FUNCTION_BLOCK EM_LiftingTransport EXTENDS EM_Base IMPLEMENTS I_EM_LiftingTransport

VAR_INPUT
//Inputs
	i_ref_stSettings : REFERENCE TO ST_SettingsLiftingTransport;
	
	i_bIlckLiftUp : BOOL := TRUE;
	i_bIlckLiftDown : BOOL := TRUE;
	i_bIlckTransportExtract : BOOL := TRUE;
	i_bIlckTransportRetract : BOOL := TRUE;
	
	i_refTB : REFERENCE TO OBJ_Carrier;	//Mogelijk voor uiteindelijke machine, voor de FUMO's is dit nog niet echt relevant
	
	
	s_arr_bTest : ARRAY[0..15] OF BOOL; 
END_VAR

VAR_OUTPUT
	q_bStaWarning : BOOL;
END_VAR

VAR
	
axisLift : AXIS_REF;
axisTransportUnit : AXIS_REF;

//------------------------------------------//
//Control Modules (Devices)
	s_cmLift : CM_AX5000;
	s_cmTransportUnit : CM_AX5000;
	
//------------------------------------------//

//------------------------------------------//
//Inputs
//------------------------------------------//
	
//------------------------------------------//
//Outputs

//------------------------------------------//

//Requests
{warning '#TODO": Update to Lifting Transport'}
s_bReqTB_ToInfeed : BOOL := FALSE;
s_bReqTB_ToCenter : BOOL := FALSE;
s_bReqTB_ToDocking : BOOL := FALSE;
s_bReqCenteringTB : BOOL := FALSE;

//States
{warning '#TODO": Update to Lifting Transport'}
s_bStaBrakeReleased : BOOL := FALSE;
s_bStaDriveError : BOOL := FALSE;

//Properties
	
//Interlockes	
	s_bIlckLiftUp : BOOL := TRUE;
	s_bIlckLiftDown : BOOL := TRUE;
	s_bIlckTransportExtract : BOOL := TRUE;
	s_bIlckTransportRetract : BOOL := TRUE;
	
	{warning '#TODO: are these variable / properies really nessecary?' }
	s_bStaTB_AtInfeed : BOOL;
	s_bStaTB_AtCentering : BOOL;
	s_bStaTB_AtDocking : BOOL;
	s_bStaTB_CenteringDone : BOOL;
	
	
//Alarms
	s_sReason : STRING;
	{warning '#TODO": Update to Lifting Transport'}
	s_fbAlarmHandlerTravelTimeOut : FB_AlarmHandler;
	s_bErrTravelTimeOut : BOOL;
	
//Warnings
{warning '#TODO": Update to Lifting Transport'}
	s_fbAlarmHandlerOuterDoorNotOpened : FB_AlarmHandler;
	s_bWrnOuterDoorNotOpened : BOOL;
	
	s_bStaWarning : BOOL;
	
//------------------------------------------//
//Params
//--	//Tool settings
//--	s_fbParamToolHardwareNr				: FB_HmiParamHandler;
//--    s_fbParamToolSoftwareVersion		: FB_HmiParamHandler;

//--	s_fbParamName						: FB_HmiParamHandler;
//--	s_fbParamNumber						: FB_HmiParamHandler;
//--	s_fbParamRevision                   : FB_HmiParamHandler;
	
//--	s_fbParamTeslaMeterIp				: FB_HmiParamHandler;
//--	s_fbParamTeslaMeterPort				: FB_HmiParamHandler;
	
//--	//Product settings (Maybe)
//--	s_fbParamTotalStroke				: FB_HmiParamHandler;
//--	s_fbParamStepStroke					: FB_HmiParamHandler;
//--	s_fbParamAveragingNumberTest		: FB_HmiParamHandler;
	
//--	s_fbParamaMaxMagnitudeCriteria		: FB_HmiParamHandler;
	
//--	s_fbParamRefIduBottom				: FB_HmiParamHandler;
//--	s_fbParamRefItm                     : FB_HmiParamHandler;
//--	s_fbParamRefCenterTpmPipe           : FB_HmiParamHandler;
//--	s_fbParamRefCpValve					: FB_HmiParamHandler;
//------------------------------------------//

//------------------------------------------//
//Variables
//--	s_sTestResult 						: STRING;
	
//------------------------------------------//

//------------------------------------------//
//Alarms
	

//------------------------------------------//

//------------------------------------------//

	s_sMessage : STRING;

//Sequencers
	s_eSeqLiftingTransport : E_SeqLiftingTransport;
	s_fbSeqLiftingTransportControl : FB_SeqControl;

	s_eTmpLocation : E_Location;
	s_eTmpCenteringDone : BOOL;
	
	s_tMaxTravelTime : TIME;
	s_tDoorCheckTime : TIME;
	s_bDoorCheckTimeDisabled : BOOL := FALSE;
	

//Hmi
{warning '#TODO": Update to Lifting Transport'}
	s_nToHmiStepNr					: INT;
	s_nToHmiMaxStepNr				: INT;
	s_sToHmiInstructionText			: T_MAXSTRING;
	s_sToHmiProcedure				: T_MAXSTRING;
	
	//Buttons
	s_fbHmiBtnTB_ToInfeed				: FB_HmiBtn;
	s_fbHmiBtnTB_ToCentering			: FB_HmiBtn;
	s_fbHmiBtnTB_ToDocking				: FB_HmiBtn;
	
	s_fbHmiBtnTB_Centering				: FB_HmiBtn;
	
	//Leds
	s_fbHmiLedInfeedRearPosition		: FB_HmiLed;
	s_fbHmiLedInfeedFrontPosition		: FB_HmiLed;
	s_fbHmiLedCenteringPosition			: FB_HmiLed;
	s_fbHmiLedDockingPosition			: FB_HmiLed;
	s_fbHmiLedDoorOpened				: FB_HmiLed;
	
	s_fbHmiLedCenteringIdle				: FB_HmiLed;
	s_fbHmiLedCenteringCenter			: FB_HmiLed;
	
//------------------------------------------//
END_VAR

	
SUPER^();

METHOD PROTECTED _m_Alarms : BOOL

IF NOT SUPER^._m_Alarms() THEN
	RETURN;
END_IF

{warning '#TODO": Update to Lifting Transport'}
// Alarm Handlers
s_fbAlarmHandlerTravelTimeOut(
	i_bStaActive := s_bErrTravelTimeOut, 
	i_eAlarmLevel := E_AlarmLevel.Alarm, 
	i_sAlarmText := CONCAT(i_sEmName, CONCAT( ': Travel error: ', s_sReason)));
	
s_fbAlarmHandlerOuterDoorNotOpened(
	i_bStaActive := s_bWrnOuterDoorNotOpened, 
	i_eAlarmLevel := E_AlarmLevel.Warning, 
	i_sAlarmText := CONCAT(i_sEmName, ': Outer-door open not detected'));

// Reset warnings
IF i_bCmdReset THEN
	s_bErrTravelTimeOut := FALSE;
	s_bWrnOuterDoorNotOpened := FALSE;
END_IF

s_bStaError := 
	s_cmPalletConveyor.p_bStaError
	OR s_cmCenteringUnit.p_bStaError
	OR s_fbAlarmHandlerTravelTimeOut.q_bStaActive;	

s_bStaWarning :=
	s_fbAlarmHandlerOuterDoorNotOpened.q_bStaActive
	OR s_cmPalletConveyor.p_bStaWarning
	OR s_cmCenteringUnit.p_bStaWarning;
	
_m_Alarms := TRUE;
END_METHOD

METHOD PRIVATE _m_AutomaticControl : BOOL

//Lifting Transport
_m_SeqLiftingTransport();
END_METHOD

METHOD PROTECTED _m_Devices : BOOL

IF NOT SUPER^._m_Devices() THEN
	RETURN;
END_IF

s_cmLift(
	i_bReqEnable := i_bReqEnable,
	i_eCtrlMode := i_eCtrlMode,
	i_bCmdReset := i_bCmdReset,
	i_refAxis := axisLift,
	i_bIclkForward := FALSE,
	i_bIclkBackward := FALSE);

s_cmTransportUnit(
	i_bReqEnable := i_bReqEnable,
	i_eCtrlMode := i_eCtrlMode,
	i_bCmdReset := i_bCmdReset,
	i_refAxis := axisTransportUnit,
	i_bIclkForward := FALSE, 
	i_bIclkBackward := FALSE);

_m_Devices := TRUE;
END_METHOD

METHOD PROTECTED _m_Hmi : BOOL

IF NOT SUPER^._m_Hmi() THEN
	RETURN;
END_IF

//Buttons
s_fbHmiBtnTB_ToInfeed.p_bStaEnabled := s_bIlckConveyorBackward;
s_fbHmiBtnTB_ToCentering.p_bStaEnabled := s_bIlckConveyorForward;
s_fbHmiBtnTB_ToDocking.p_bStaEnabled := s_bIlckConveyorForward;
s_fbHmiBtnTB_Centering.p_bStaEnabled := s_bIlckCenteringToCenter;

s_fbHmiBtnTB_ToInfeed();
s_fbHmiBtnTB_ToCentering();
s_fbHmiBtnTB_ToDocking();
s_fbHmiBtnTB_Centering();

//Leds
s_fbHmiLedInfeedRearPosition(i_bStaLed := s_bStaAtInfeedRearPosition);
s_fbHmiLedInfeedFrontPosition(i_bStaLed := s_bStaAtInfeedFrontPosition);
s_fbHmiLedCenteringPosition(i_bStaLed := s_bStaAtCenteringPosition);
s_fbHmiLedDockingPosition(i_bStaLed := s_bStaAtDockingPosition);
s_fbHmiLedDoorOpened(i_bStaLed := s_bStaDoorOpened);

s_fbHmiLedCenteringCenter(i_bStaLed := s_bStaCenteringCenter);
s_fbHmiLedCenteringIdle(i_bStaLed := s_bStaCenteringIdle);

_m_Hmi := TRUE;
END_METHOD

METHOD PROTECTED _m_Init : BOOL

IF NOT SUPER^._m_Init() THEN
	RETURN;
END_IF

//Control Modules
s_cmLift.i_bReqEnable := FALSE;
s_cmLift.i_eCtrlMode := E_CtrlMode.IDLE;
s_cmLift.i_sCmName := 'CM Lift';
s_cmLift.i_refAxis REF= axisLift;

s_cmTransportUnit.i_bReqEnable := FALSE;
s_cmTransportUnit.i_eCtrlMode := E_CtrlMode.IDLE;
s_cmTransportUnit.i_sCmName := 'CM Transport Unit';
s_cmTransportUnit.i_refAxis REF= axisTransportUnit;
{warning '#TODO: Dot we need to added configuration parameters? Seperate struct or via settings or dedicateed variables'}

//---------------------------------//	
	
//----------------------------------//	
//Hmi
{warning '#TODO: Update to Lifing Transport'} 
	s_fbHmiBtnTB_ToInfeed.p_eButtontype := E_HmiButtonType.PUSHBUTTON;
	s_fbHmiBtnTB_ToInfeed.p_bStaVisible := FALSE;
	s_fbHmiBtnTB_ToInfeed.p_bStaEnabled := FALSE;		
	s_fbHmiBtnTB_ToInfeed.p_sBtnText := 'TB To Infeed Position';
	
	s_fbHmiBtnTB_ToCentering.p_eButtontype := E_HmiButtonType.PUSHBUTTON;
	s_fbHmiBtnTB_ToCentering.p_bStaVisible := FALSE;
	s_fbHmiBtnTB_ToCentering.p_bStaEnabled := FALSE;		
	s_fbHmiBtnTB_ToCentering.p_sBtnText := 'TB To Centering Position';
	
	s_fbHmiBtnTB_ToDocking.p_eButtontype := E_HmiButtonType.PUSHBUTTON;
	s_fbHmiBtnTB_ToDocking.p_bStaVisible := FALSE;
	s_fbHmiBtnTB_ToDocking.p_bStaEnabled := FALSE;		
	s_fbHmiBtnTB_ToDocking.p_sBtnText := 'TB To Docking Position';
	
	s_fbHmiBtnTB_Centering.p_eButtontype := E_HmiButtonType.PUSHBUTTON;
	s_fbHmiBtnTB_Centering.p_bStaVisible := FALSE;
	s_fbHmiBtnTB_Centering.p_bStaEnabled := FALSE;		
	s_fbHmiBtnTB_Centering.p_sBtnText := 'Centering TB';

	s_fbHmiLedInfeedRearPosition.p_bStaVisible := FALSE;
	s_fbHmiLedInfeedRearPosition.p_sToHmiDescriptionLed := 'Infeed Rear Position';
	
	s_fbHmiLedInfeedFrontPosition.p_bStaVisible := FALSE;
	s_fbHmiLedInfeedFrontPosition.p_sToHmiDescriptionLed := 'Infeed Front Position';
	
	s_fbHmiLedCenteringPosition.p_bStaVisible := FALSE;
	s_fbHmiLedCenteringPosition.p_sToHmiDescriptionLed := 'Center Position';
	
	s_fbHmiLedDockingPosition.p_bStaVisible := FALSE;
	s_fbHmiLedDockingPosition.p_sToHmiDescriptionLed := 'Docking Position';
	
	s_fbHmiLedDoorOpened.p_bStaVisible := FALSE;
	s_fbHmiLedDoorOpened.p_sToHmiDescriptionLed := 'Door Opened';
	
	s_fbHmiLedCenteringIdle.p_bStaVisible := FALSE;
	s_fbHmiLedCenteringIdle.p_sToHmiDescriptionLed := 'Centering Idle';
	
	s_fbHmiLedCenteringCenter.p_bStaVisible := FALSE;
	s_fbHmiLedCenteringCenter.p_sToHmiDescriptionLed := 'Centering Center';
	
//----------------------------------//	
//Initialize all moving averages

//----------------------------------//	

//----------------------------------//	

//Inputs
//----------------------------------//	

//----------------------------------//	
//Outputs
//--s_doRelayTableDown.i_stSettings.bCfgDelay		:= FALSE;	
//--s_doRelayTableDown.i_stSettings.tmOutputDelay	:= T#0S;	
//----------------------------------//	

_m_Init := TRUE;
END_METHOD

METHOD PROTECTED _m_Inputs : BOOL
IF NOT SUPER^._m_Inputs() THEN
	RETURN;
END_IF

//Interlocks
s_bIlckConveyorForward := i_bIlckConveyorForward OR NOT(s_bStaCenteringIdle); 
s_bIlckConveyorBackward := i_bIlckConveyorBackward OR NOT(s_bStaCenteringIdle);
s_bIlckConveyorBackward := NOT(s_bStaCenteringIdle);
s_bIlckCenteringToCenter := NOT(s_cmPalletConveyor.p_bStaMotorStopped);
s_bIlckCenteringToIdle := FALSE;

//Reasons
IF i_bIlckConveyorForward OR i_bIlckConveyorBackward THEN
	s_cmPalletConveyor.p_sInterlockedReason := 'External interlocked';
ELSIF s_bIlckConveyorForward OR s_bIlckConveyorBackward THEN
	s_cmPalletConveyor.p_sInterlockedReason := 'Centering not in idle-position'; 
END_IF

IF s_bIlckCenteringToCenter THEN
	s_cmCenteringUnit.p_sInterlockedReason := 'Conveyor not stopped';
END_IF

_m_Inputs := TRUE;
END_METHOD

METHOD PRIVATE _m_ManualControl : BOOL

// Manual control has been implemented into lower layer control modules
END_METHOD

METHOD _m_MoveAbsolute : BOOL
VAR_INPUT
	i_ref_axis : REFERENCE TO TC2_MC2.AXIS_REF;
	i_ref_stProfile : ST_PositioningProfile;
END_VAR

VAR_INST
	s_MC_MoveAbsolute : TC2_MC2.MC_MoveAbsolute;
END_VAR

IF NOT(__ISVALIDREF(i_ref_axis)) THEN
	// Message invalid reference
	RETURN;
END_IF

s_MC_MoveAbsolute(
	Axis := i_ref_axis,
	Execute := TRUE AND NOT(s_MC_MoveAbsolute.Busy OR s_MC_MoveAbsolute.Done OR s_MC_MoveAbsolute.Error),
	Position := i_ref_stProfile.fPosition,
	Velocity := i_ref_stProfile.fVelocity,
	Acceleration := i_ref_stProfile.fAcceleration,
	Deceleration := i_ref_stProfile.fDeceleration,
	Jerk := i_ref_stProfile.fJerk,
	BufferMode := TC2_MC2.MC_BufferMode.MC_Aborting,
	Options := ,
	Done => ,
	Busy => ,
	Active => ,
	CommandAborted => ,
	Error => ,
	ErrorID => );
	
_m_MoveAbsolute := s_MC_MoveAbsolute.Done;
END_METHOD

METHOD PROTECTED _m_Outputs : BOOL

IF NOT SUPER^._m_Outputs() THEN
	RETURN;
END_IF

q_bStaWarning := s_bStaWarning;

_m_Outputs := TRUE;
END_METHOD

METHOD PROTECTED _m_Params : BOOL
VAR_INST
	s_fToHmiXAxisMin	: LREAL;
	s_fToHmiXAxisMax	: LREAL;
	s_fToHmiYAxisMin	: LREAL;
	s_fToHmiYAxisMax	: LREAL;
END_VAR

IF NOT SUPER^._m_Params() THEN
	RETURN;
END_IF

s_fbParamToolHardwareNr(i_fDefaultValue				:= 0,
						i_nArrayFolderIndex			:= 1,
						i_sName						:= 'Harware ID',
						i_bIsNumber					:= FALSE);

s_fbParamToolSoftwareVersion(i_fDefaultValue		:= 0,
							i_nArrayFolderIndex		:= 1,
							i_sName					:= 'Software Version',
							i_bIsNumber				:= FALSE);

s_fbParamName(i_fDefaultValue						:= 0,
				i_nArrayFolderIndex					:= 1,
				i_sName								:= 'Description',
				i_bIsNumber							:= FALSE);
							
s_fbParamTeslaMeterIp(i_fDefaultValue			:= 0,
						i_nArrayFolderIndex		:= 1,
						i_sName					:= 'Tesla meter ip adress',
						i_bIsNumber				:= FALSE);
						
s_fbParamTeslaMeterPort(i_fDefaultValue			:= 0,
						i_nArrayFolderIndex		:= 1,
						i_sName					:= 'Tesla meter port number',
						i_bIsNumber				:= TRUE);

//---------

						
s_fbParamTotalStroke(i_fDefaultValue			:= 100,
						i_nArrayFolderIndex		:= 2,
						i_sName					:= 'Total measurement stroke',
						i_bIsNumber				:= TRUE);
						
s_fbParamStepStroke(i_fDefaultValue				:= 10,
						i_nArrayFolderIndex		:= 2,
						i_sName					:= 'Step distance per measurement',
						i_bIsNumber				:= TRUE);

s_fbParamAveragingNumberTest(i_fDefaultValue		:= 10,
							i_nArrayFolderIndex		:= 2,
							i_sName					:= 'Number of measurements per step for averaging the magnetic field',
							i_bIsNumber				:= TRUE);
							
s_fbParamaMaxMagnitudeCriteria(i_fDefaultValue		:= 100,
							i_nArrayFolderIndex		:= 2,
							i_sName					:= 'Maximum allowed magnitude magnetic field (Test)',
							i_bIsNumber				:= TRUE);

s_fbParamRefIduBottom(i_fDefaultValue				:= 0,
							i_nArrayFolderIndex		:= 2,
							i_sName					:= 'Distance from home position to lower IDU Bottom',
							i_bIsNumber				:= TRUE);
							
s_fbParamRefItm(i_fDefaultValue						:= 0,
							i_nArrayFolderIndex		:= 2,
							i_sName					:= 'Distance from home position Itm lower IDU / upper IDU',
							i_bIsNumber				:= TRUE);
							
s_fbParamRefCenterTpmPipe(i_fDefaultValue			:= 0,
							i_nArrayFolderIndex		:= 2,
							i_sName					:= 'Distance from home position to center TPM pipe',
							i_bIsNumber				:= TRUE);
							
s_fbParamRefCpValve(i_fDefaultValue		:= 0,
							i_nArrayFolderIndex		:= 2,
							i_sName					:= 'Distance from home position to bottom C/P valve',
							i_bIsNumber				:= TRUE);				

GVL_DataLogging.g_stReportData.CabinetSerialNumber      := s_fbParamToolHardwareNr.p_sValue;
GVL_DataLogging.g_stReportData.TesterSoftwareVersion    := s_fbParamToolSoftwareVersion.p_sValue;
GVL_DataLogging.g_stReportData.Operator                 := GVL.g_sUser;
GVL_DataLogging.g_stReportData.Note						:= GVL.g_sNotesEntry;
//GVL_DataLogging.g_stReportData.Message can be filled in test procedure with for example the error if test is stopped
GVL_DataLogging.g_stReportData.SerialNumber             := GVL.g_sSerialNumber;

s_fToHmiXAxisMin	:= -2*s_fbParamaMaxMagnitudeCriteria.p_fValue;
s_fToHmiXAxisMax	:= 2*s_fbParamaMaxMagnitudeCriteria.p_fValue;
s_fToHmiYAxisMin	:= s_CmProbeMotor.p_fHomePosition;
s_fToHmiYAxisMax	:= s_fbParamRefCpValve.p_fValue*1.2;

_m_Params := TRUE;
END_METHOD

METHOD PRIVATE _m_SeqLiftingTransport : BOOL

s_fbHmiBtnTB_ToInfeed.p_bStaVisible := TRUE;
//--s_fbHmiBtnTB_ToInfeed.p_bStaEnabled := TRUE;

s_fbHmiBtnTB_ToCentering.p_bStaVisible := TRUE;
//--s_fbHmiBtnTB_ToCentering.p_bStaEnabled := TRUE;

s_fbHmiBtnTB_ToDocking.p_bStaVisible := TRUE;
//--s_fbHmiBtnTB_ToDocking.p_bStaEnabled := TRUE;

s_fbSeqLiftingTransportControl(
	i_nSeqStep := s_eSeqLiftingTransport, 
	i_sStepName := TO_STRING(s_eSeqLiftingTransport), 
	i_bCmdReset := i_bCmdReset
					AND (s_eSeqLiftingTransport = E_SeqTransport.ERROR) // Only reset/resume sequencer from ERROR state
					AND NOT(s_cmLift.p_bStaError)
					AND NOT(s_cmTransportUnit.p_bStaError)
					AND i_bReqEnable, 
	i_bStaError := s_bStaError OR NOT(i_bReqEnable) AND FALSE);
	
CASE s_eSeqLiftingTransport OF
	
	E_SeqLiftingTransport.IDLE:
		s_eTmpLocation := E_Location.UNKNOWN;
	
		
		
		s_eSeqLiftingTransport := E_SeqLiftingTransport.START;
		
	E_SeqLiftingTransport.START:
		//--IF s_fbSeqTransportControl.q_tmStepTime > T#1S THEN
		//--	s_eSeqTransport := E_SeqTransport.READY;
		//--END_IF
		
		IF s_fbSeqLiftingTransportControl.q_bStaEntry THEN
			;//--s_cmPalletConveyor.m_Stop();
		END_IF		
	
		//IF s_cmPalletConveyor.p_bStaMotorStopped AND_THEN NOT(s_cmPalletConveyor.p_bStaBrakeReleased) AND s_fbSeqTransportControl.q_tmStepTime > T#1S THEN
		//	s_eSeqLiftingTransport := E_SeqTransport.READY;
		//END_IF
		
		s_cmLift.m_MC_Power(
			i_bEnable := TRUE,
			i_bEnablePositive := TRUE,
			i_bEnableNegative := TRUE,
			i_fOverride := 100.0,
			i_eBufferMode := TC2_MC2.MC_BufferMode.MC_Aborting);
			
		s_cmTransportUnit.m_MC_Power(
			i_bEnable := TRUE,
			i_bEnablePositive := TRUE,
			i_bEnableNegative := TRUE,
			i_fOverride := 100.0,
			i_eBufferMode := TC2_MC2.MC_BufferMode.MC_Aborting);
		
		IF s_arr_bTest[0] THEN
			s_arr_bTest[0] := FALSE;
			s_eSeqLiftingTransport := E_SeqLiftingTransport.LIFT_PRE_PICK_TROLLEY_IN_TB;
		END_IF
	
	E_SeqLiftingTransport.HOME_TRANSPORT:
		IF s_fbSeqLiftingTransportControl.q_bStaEntry THEN
			s_cmTransportUnit.m_MC_Home(
				i_bExecute := TRUE,
				i_fPosition := 0.0,
				i_eHomingMode := Tc2_MC2.MC_HomingMode.MC_Direct,
				i_eBufferMode := Tc2_MC2.MC_BufferMode.MC_Aborting);
		END_IF
		
		IF s_cmTransportUnit.p_bDone THEN
			s_eSeqLiftingTransport := E_SeqLiftingTransport.HOME_LIFT;
		ELSIF s_cmTransportUnit.p_bError THEN
			s_eSeqLiftingTransport := E_SeqLiftingTransport.ERROR;
		ELSIF s_fbSeqLiftingTransportControl.q_tmStepTime > T#30S THEN
			s_eSeqLiftingTransport := E_SeqLiftingTransport.ERROR;
		END_IF	
	
	E_SeqLiftingTransport.HOME_LIFT:
		IF s_fbSeqLiftingTransportControl.q_bStaEntry THEN
			s_cmLift.m_MC_Home(
				i_bExecute := TRUE,
				i_fPosition := 0.0,
				i_eHomingMode := Tc2_MC2.MC_HomingMode.MC_Direct,
				i_eBufferMode := Tc2_MC2.MC_BufferMode.MC_Aborting);
		END_IF
		
		IF s_cmLift.p_bDone THEN
			s_eSeqLiftingTransport := E_SeqLiftingTransport.HOME_LIFT;
		ELSIF s_cmLift.p_bError THEN
			s_eSeqLiftingTransport := E_SeqLiftingTransport.ERROR;
		ELSIF s_fbSeqLiftingTransportControl.q_tmStepTime > T#30S THEN
			s_eSeqLiftingTransport := E_SeqLiftingTransport.ERROR;
		END_IF		
	
	E_SeqLiftingTransport.MOVE_TO_IDLE:
	
/// PICK TROLLEY IN TB /////////////////////////////////////////////////////////
	E_SeqLiftingTransport.LIFT_PRE_PICK_TROLLEY_IN_TB:
		IF _m_MoveAbsolute(	i_ref_AXIS := axisLift, i_ref_stProfile := i_ref_stSettings.arr_LiftPositioningProfile[1]) THEN
			s_eSeqLiftingTransport := E_SeqLiftingTransport.TRANSPORT_PRE_PICK_TROLLEY_IN_TB;
		END_IF
	
	E_SeqLiftingTransport.TRANSPORT_PRE_PICK_TROLLEY_IN_TB:
		IF _m_MoveAbsolute(	i_ref_AXIS := axisTransportUnit, i_ref_stProfile := i_ref_stSettings.arr_TransportUnitPositioningProfile[1]) THEN
			s_eSeqLiftingTransport := E_SeqLiftingTransport.TRANSPORT_PICK_TROLLEY_IN_TB;
		END_IF
	
	E_SeqLiftingTransport.TRANSPORT_PICK_TROLLEY_IN_TB:
		IF _m_MoveAbsolute(	i_ref_AXIS := axisTransportUnit, i_ref_stProfile := i_ref_stSettings.arr_TransportUnitPositioningProfile[2]) THEN
			s_eSeqLiftingTransport := E_SeqLiftingTransport.LIFT_PICK_TROLLEY_IN_TB;
		END_IF
	
	E_SeqLiftingTransport.LIFT_PICK_TROLLEY_IN_TB:
		IF _m_MoveAbsolute(	i_ref_AXIS := axisLift, i_ref_stProfile := i_ref_stSettings.arr_LiftPositioningProfile[2]) THEN
			s_eSeqLiftingTransport := E_SeqLiftingTransport.LIFT_RAISE_TROLLEY_IN_TB;
		END_IF
	
	E_SeqLiftingTransport.LIFT_RAISE_TROLLEY_IN_TB:
		IF _m_MoveAbsolute(	i_ref_AXIS := axisLift, i_ref_stProfile := i_ref_stSettings.arr_LiftPositioningProfile[3]) THEN
			s_eSeqLiftingTransport := E_SeqLiftingTransport.TRANSPORT_PLACE_TROLLEY_IN_CABIN;
		END_IF

/// PLACE TROLLEY IN TB ////////////////////////////////////////////////////////	
	E_SeqLiftingTransport.TRANSPORT_PLACE_TROLLEY_IN_CABIN:
		IF _m_MoveAbsolute(	i_ref_AXIS := axisTransportUnit, i_ref_stProfile := i_ref_stSettings.arr_TransportUnitPositioningProfile[3]) THEN
			s_eSeqLiftingTransport := E_SeqLiftingTransport.LIFT_PRE_PLACE_TROLLEY_IN_CABIN;
		END_IF
		
	E_SeqLiftingTransport.LIFT_PRE_PLACE_TROLLEY_IN_CABIN:
		IF _m_MoveAbsolute(	i_ref_AXIS := axisLift, i_ref_stProfile := i_ref_stSettings.arr_LiftPositioningProfile[4]) THEN
			s_eSeqLiftingTransport := E_SeqLiftingTransport.LIFT_PLACE_TROLLEY_IN_CABIN;
		END_IF
		
	E_SeqLiftingTransport.LIFT_PLACE_TROLLEY_IN_CABIN:
		IF _m_MoveAbsolute(	i_ref_AXIS := axisLift, i_ref_stProfile := i_ref_stSettings.arr_LiftPositioningProfile[5]) THEN
			s_eSeqLiftingTransport := E_SeqLiftingTransport.LIFT_PRE_PICK_TROLLEY_IN_CABIN;
		END_IF

/// PICK TROLLEY IN CABIN //////////////////////////////////////////////////////		
	E_SeqLiftingTransport.LIFT_PRE_PICK_TROLLEY_IN_CABIN:
		IF _m_MoveAbsolute(	i_ref_AXIS := axisLift, i_ref_stProfile := i_ref_stSettings.arr_LiftPositioningProfile[6]) THEN
			s_eSeqLiftingTransport := E_SeqLiftingTransport.LIFT_PICK_TROLLEY_IN_CABIN;
		END_IF
		
	E_SeqLiftingTransport.LIFT_PICK_TROLLEY_IN_CABIN:
		IF _m_MoveAbsolute(	i_ref_AXIS := axisLift, i_ref_stProfile := i_ref_stSettings.arr_LiftPositioningProfile[7]) THEN
			s_eSeqLiftingTransport := E_SeqLiftingTransport.LIFT_RAISE_TROLLEY_IN_CABIN;
		END_IF
		
	E_SeqLiftingTransport.LIFT_RAISE_TROLLEY_IN_CABIN:
		IF _m_MoveAbsolute(	i_ref_AXIS := axisLift, i_ref_stProfile := i_ref_stSettings.arr_LiftPositioningProfile[8]) THEN
			s_eSeqLiftingTransport := E_SeqLiftingTransport.TRANSPORT_PRE_PLACE_TROLLEY_IN_TB;
		END_IF
	
/// PLACE TROLLEY IN TB //??////////////////////////////////////////////////////
	E_SeqLiftingTransport.TRANSPORT_PRE_PLACE_TROLLEY_IN_TB:
		IF _m_MoveAbsolute(	i_ref_AXIS := axisTransportUnit, i_ref_stProfile := i_ref_stSettings.arr_TransportUnitPositioningProfile[4]) THEN
			s_eSeqLiftingTransport := E_SeqLiftingTransport.TRANSPORT_PLACE_TROLLEY_IN_TB;
		END_IF
	
	E_SeqLiftingTransport.TRANSPORT_PLACE_TROLLEY_IN_TB:
		IF _m_MoveAbsolute(	i_ref_AXIS := axisTransportUnit, i_ref_stProfile := i_ref_stSettings.arr_TransportUnitPositioningProfile[5]) THEN
			s_eSeqLiftingTransport := E_SeqLiftingTransport.LIFT_PRE_PLACE_TROLLEY_IN_TB;
		END_IF

	E_SeqLiftingTransport.LIFT_PRE_PLACE_TROLLEY_IN_TB:
		IF _m_MoveAbsolute(	i_ref_AXIS := axisLift, i_ref_stProfile := i_ref_stSettings.arr_LiftPositioningProfile[9]) THEN
			s_eSeqLiftingTransport := E_SeqLiftingTransport.LIFT_PLACE_TROLLEY_IN_TB;
		END_IF
		
	E_SeqLiftingTransport.LIFT_PLACE_TROLLEY_IN_TB:
		IF _m_MoveAbsolute(	i_ref_AXIS := axisLift, i_ref_stProfile := i_ref_stSettings.arr_LiftPositioningProfile[10]) THEN
			s_eSeqLiftingTransport := E_SeqLiftingTransport.START;
		END_IF
		
	E_SeqLiftingTransport.READY:
		IF s_fbSeqLiftingTransportControl.q_bStaEntry THEN
			i_refTB.p_eLocation := s_eTmpLocation;
			s_eTmpLocation := E_Location.UNKNOWN;
		END_IF
		
(*		i_refTB.p_bOuterDoorOpened S= s_bStaAtInfeedRearPosition AND s_bStaAtInfeedFrontPosition AND s_bStaDoorOpened;
	
		IF s_fbHmiBtnTB_ToInfeed.p_osrBtnPress OR s_bReqTB_ToInfeed THEN
			IF m_CmdTB_ToInfeed(o_sReason => s_sMessage) THEN
				s_eSeqTransport := E_SeqTransport.MOVE_TO_INFEED;
			ELSE	
				//Write message
				//--s_sMessage := m_TB_ToCenter.o_sReason;
			END_IF
 
			s_bReqTB_ToInfeed := FALSE;
			
			//--AND NOT(s_bStaAtInfeedRearPosition)
			//--THEN
			
		ELSIF s_fbHmiBtnTB_ToCentering.p_osrBtnPress OR s_bReqTB_ToCenter THEN
			IF m_CmdTB_ToCenter(o_sReason => s_sMessage) THEN
				s_eSeqTransport := E_SeqTransport.MOVE_TO_CENTERING;
			ELSE	
				//Write message
				//--s_sMessage := m_TB_ToCenter.o_sReason;
			END_IF	
		
			s_bReqTB_ToCenter := FALSE;
			
			//--AND NOT(s_bStaAtCenteringPosition)
			//--THEN
			
			//--IF s_bStaDoorOpened THEN
			//--	s_eSeqTransport := E_SeqTransport.MOVE_TO_Centering;
			//--ELSE
			//--	s_bWrnOuterDoorNotOpened := TRUE;
			//--END_IF
			
		ELSIF s_fbHmiBtnTB_ToDocking.p_osrBtnPress OR s_bReqTB_ToDocking THEN
			IF m_CmdTB_ToDocking(o_sReason => s_sMessage) THEN
				s_eSeqTransport := E_SeqTransport.MOVE_TO_DOCKING;
			ELSE	
				//Write message
				//--s_sMessage := m_TB_ToDocking.o_sReason;
			END_IF	
		
			s_bReqTB_ToDocking := FALSE;
			
		//--	AND NOT(s_bStaAtDockingPosition)
		//--	THEN
		//--	s_eSeqTransport := E_SeqTransport.MOVE_TO_DOCKING;
		END_IF	
	
	E_SeqTransport.MOVE_TO_INFEED:
		IF s_fbSeqTransportControl.q_bStaEntry THEN		
			s_tMaxTravelTime := LREAL_TO_TIME((i_ref_stSettings.fDistanceToInfeed / i_ref_stSettings.fSpeedGoToInfeed) * i_ref_stSettings.fTravelTollerance * 1000);
			s_cmPalletConveyor.m_StartBackward(i_rTargetSpeed := i_stSettings.fSpeedGoToInfeed);
		END_IF
		
		IF s_bStaAtInfeedRearPosition THEN
			s_eTmpLocation := E_Location.INFEED;
			s_eSeqTransport := E_SeqTransport.STOP;
		ELSIF s_fbSeqTransportControl.q_tmStepTime > s_tMaxTravelTime THEN
			s_bErrTravelTimeOut := TRUE;
			s_sReason := 'Moving to infeed - timeout';
			s_eSeqTransport := E_SeqTransport.ERROR;
		END_IF
	
	E_SeqTransport.MOVE_TO_CENTERING:
		IF s_fbSeqTransportControl.q_bStaEntry THEN
			s_tMaxTravelTime := LREAL_TO_TIME((i_ref_stSettings.fDistanceToCentering / i_ref_stSettings.fSpeedGoToCentering) * i_ref_stSettings.fTravelTollerance * 1000);
			s_tDoorCheckTime := LREAL_TO_TIME((i_ref_stSettings.fDistanceOuteDoorCheck / i_ref_stSettings.fSpeedGoToCentering) * 1000);
			s_cmPalletConveyor.m_StartForward(i_rTargetSpeed := i_stSettings.fSpeedGoToCentering);
		END_IF
		
		IF s_bStaAtCenteringPosition THEN
			s_bDoorCheckTimeDisabled := FALSE;
			s_eTmpLocation := E_Location.CENTERING;
			s_eSeqTransport := E_SeqTransport.STOP;
		
		ELSIF s_fbSeqTransportControl.q_tmStepTime < s_tDoorCheckTime 
			AND NOT(s_bStaDoorOpened) THEN
			s_bWrnOuterDoorNotOpened := TRUE;
			s_bDoorCheckTimeDisabled := TRUE; //Disable error after first occurance (to prevent invalid retriggering at reties)
			s_eSeqTransport := E_SeqTransport.ERROR;
			
		ELSIF s_fbSeqTransportControl.q_tmStepTime > s_tMaxTravelTime THEN
			s_bErrTravelTimeOut := TRUE;
			s_sReason := 'Moving to Centering - timeout';
			s_eSeqTransport := E_SeqTransport.ERROR;

		//--Not clear it this will work correct due to order of sensor positions
		//--ELSIF s_bStaAtDockingPosition THEN
		//--	s_bErrTravelTimeOut := TRUE;
		//--	s_sReason := 'Moving to Centering - too far (docking)';
		//--	s_eSeqTransport := E_SeqTransport.ERROR;
		
		END_IF
	
	E_SeqTransport.MOVE_TO_DOCKING:
		IF s_fbSeqTransportControl.q_bStaEntry THEN
			s_tMaxTravelTime := LREAL_TO_TIME((i_ref_stSettings.fDistanceToDocking / i_ref_stSettings.fSpeedGoToDocking) * i_ref_stSettings.fTravelTollerance * 1000);
			s_cmPalletConveyor.m_StartForward(i_rTargetSpeed := i_stSettings.fSpeedGoToDocking);
		END_IF
		
		IF s_bStaAtDockingPosition THEN
			s_eTmpLocation := E_Location.DOCKING;
			s_eSeqTransport := E_SeqTransport.STOP;
		ELSIF s_fbSeqTransportControl.q_tmStepTime > s_tMaxTravelTime THEN
			s_bErrTravelTimeOut := TRUE;
			s_sReason := 'Moving to docking - timeout';
			s_eSeqTransport := E_SeqTransport.ERROR;		
		END_IF
		
	E_SeqTransport.STOP:
		IF s_fbSeqTransportControl.q_bStaEntry THEN
			s_cmPalletConveyor.m_Stop();
		END_IF
		
		IF s_cmPalletConveyor.p_bStaMotorStopped THEN
			s_eSeqTransport := E_SeqTransport.READY;
		END_IF
		
	E_SeqTransport.ERROR:
		s_cmPalletConveyor.m_Stop();
*)		
END_CASE
END_METHOD

METHOD PUBLIC m_CmdCenteringTB : BOOL
VAR_INPUT
	i_refReason : REFERENCE TO STRING;
END_VAR
VAR_OUTPUT
	o_sReason : STRING;
END_VAR

IF NOT i_bReqEnable THEN 
	RETURN;
END_IF

//--IF NOT(s_bIlckCenteringToCenter) THEN
//--	s_bReqCenteringTB := TRUE;
//--	m_CenteringTB := TRUE;
//--ELSE
//--	m_CenteringTB := FALSE;	
//--END_IF

IF s_bIlckCenteringToCenter THEN
	i_refReason := 'Command Centering: Interlocked';
	m_CmdCenteringTB := FALSE;
ELSE
	m_CmdCenteringTB := TRUE;	
END_IF
END_METHOD

METHOD PUBLIC m_CmdTB_ToCenter : BOOL
VAR_OUTPUT
	o_sReason : STRING;
END_VAR

IF NOT i_bReqEnable THEN 
	RETURN;
END_IF

//--IF NOT(s_bIlckConveyorForward) 
//--	AND NOT(s_bStaAtCenteringPosition)
//--	THEN
//--	s_bReqTB_ToCenter := TRUE;
//--	m_TB_ToCenter := TRUE;
//--ELSE
//--	m_TB_ToCenter := FALSE;	
//--END_IF

////////

IF s_bIlckConveyorForward THEN
	o_sReason := 'Command To Center: Interlocked';
	m_CmdTB_ToCenter := FALSE;
ELSIF s_bStaAtCenteringPosition THEN
 	o_sReason := 'Already at center position';
	m_CmdTB_ToCenter := FALSE;
ELSIF NOT(s_bStaDoorOpened) THEN
	o_sReason := 'Door not opened';
	s_bWrnOuterDoorNotOpened := TRUE; // kan mogelijk vervallen wanneer er toch gewerkt gaat worden met reasons.
	m_CmdTB_ToCenter := FALSE;
ELSE
	m_CmdTB_ToCenter := TRUE;	
END_IF
END_METHOD

METHOD PUBLIC m_CmdTB_ToDocking : BOOL
VAR_OUTPUT
	o_sReason : STRING;
END_VAR

IF NOT i_bReqEnable THEN 
	RETURN;
END_IF

//--IF NOT(s_bIlckConveyorForward) THEN
//--	s_bReqTB_ToDocking := TRUE;
//--	m_TB_ToDocking := TRUE;
//--ELSE
//--	m_TB_ToDocking := FALSE;	
//--END_IF

IF s_bStaAtDockingPosition THEN
	o_sReason := 'Command to Docking: Interlocked';
	m_CmdTB_ToDocking := FALSE;
ELSE
	m_CmdTB_ToDocking := TRUE;	
END_IF
END_METHOD

METHOD PUBLIC m_CmdTB_ToInfeed : BOOL
VAR_OUTPUT
	o_sReason : STRING;
END_VAR

IF NOT i_bReqEnable THEN 
	RETURN;
END_IF

//--IF NOT(s_bIlckConveyorBackward) 
//--	AND NOT(s_bStaAtInfeedRearPosition)
//--	THEN
//--	s_bReqTB_ToInfeed := TRUE;
//--	m_TB_ToInfeed := TRUE;
//--ELSE
//--	m_TB_ToInfeed := FALSE;	
//--END_IF

IF s_bIlckConveyorBackward THEN
	o_sReason := 'Command to Infeed: Interlocked';
	m_CmdTB_ToInfeed := FALSE;
ELSE
	m_CmdTB_ToInfeed := TRUE;	
END_IF
END_METHOD

METHOD PUBLIC m_Main : BOOL
IF NOT SUPER^.m_Main() THEN
	RETURN;
END_IF

// Pallet Conveyor
//??IF i_refTB.p_eLocation = E_Location.INFEED
//??	AND i_refTB.p_eDestination > E_Location.INFEED
//??	THEN
	
//??	s_cmPalletConveyor.m_ReleaseBrake(TRUE);

//??	IF s_cmPalletConveyor.p_bStaBrakeReleased THEN
//??		s_cmPalletConveyor.m_StartForward(i_stSettings.rSpeedGoToCentering);
//??	END_IF
	
//??END_IF

//??CASE i_refTB.p_eLocation OF
//??	E_Location.INFEED :

//??	E_Location.Centering :

//??	E_Location.DOCKING :	
		
//??		IF i_refTB.p_eDestination < E_Location.DOCKING 
//??			AND NOT(i_refTB. Docked)
//??			THEN
//??			 s_cmPalletConveyor.m_StartBackward(i_stSettings.rSpeedReturnToInfeed);
//??		END_IF

//??END_CASE


// Centering
//??IF i_refTB.p_eLocation = E_Location.Centering
//??	AND s_diStaAtCenteringPosition.p_bStaInputDelayed
//??	AND NOT(i_refTB.p_bAlligned)
//??	THEN
//??		s_cmCenteringUnit.m_On();
		
//??		IF s_cmCenteringUnit.p_bStaIsOn THEN
//??			i_refTB.p_bAlligned := TRUE;
//??		END_IF
//??ELSE
//??	s_cmCenteringUnit.m_Off();
//??END_IF

CASE i_eCtrlMode OF

	E_CtrlMode.IDLE:
	
		s_eSeqLiftingTransport := E_SeqLiftingTransport.IDLE;
		
	E_CtrlMode.AUTOMATIC:
	
		//Excecute automatic control
		_m_AutomaticControl();
		
(*		s_fbSeqDockingInterface(
			i_nSeqStep := s_eSeqDockingInterface, 
			i_sStepName := TO_STRING(s_fbSeqDockingInterface.q_eActState), 
			i_bCmdReset := i_bCmdReset, 
			i_bStaError := s_bStaError);
	
		CASE s_eSeqDockingInterface OF
			
			E_SeqDockingInterface.IDLE:
			
				IF s_bReqDockBox THEN
					//--IF s_diStaBoxAtPreDockingPosition.p_bStaInputDelayed THEN
					IF s_bStaBoxAtPreDockingPosition THEN	
						s_bStaUndockingDone := FALSE;
						s_eSeqDockingInterface := E_SeqDockingInterface.DOCKING_CLOSE_CLAMPS;
					ELSE
						s_bWrnNoBoxPresentAtPreDockingPosition := TRUE;	
					END_IF
				END_IF
				
				IF s_bReqUndockBox THEN
					IF s_diStaBoxAtDockedPosition.p_bStaInputDelayed THEN
						s_bStaDockingDone := FALSE;
						s_eSeqDockingInterface := E_SeqDockingInterface.UNDOCKING_LOCK_DOOR;
					ELSE
						s_bWrnNoBoxPresentAtDockedPosition := TRUE;	
					END_IF	
				END_IF
			
				// Seperatly opening/closing the clamps is nessescary to move these out of the way for moving of the outer door
				// Clamps must be closed before the outer door can be moved
				IF s_bReqClosDockingClamps THEN
					s_eSeqDockingInterface := E_SeqDockingInterface.ONLY_CLOSE_CLAMPS;
				END_IF
				
				IF s_bReqOpenDockingClamps THEN
					s_eSeqDockingInterface := E_SeqDockingInterface.ONLY_OPEN_CLAMPS;
				END_IF
				
			E_SeqDockingInterface.DOCKING_CLOSE_CLAMPS:
				
				IF s_fbSeqDockingInterface.q_bStaEntry THEN 
					s_cmDockingClamps.m_Close();
				END_IF
				
				IF s_cmDockingClamps.p_bStaIsClosed THEN
					s_eSeqDockingInterface := E_SeqDockingInterface.DOCKING_UNLOCK_DOOR;
				ELSIF s_cmDockingClamps.p_bStaError THEN 
					s_eSeqDockingInterface := E_SeqDockingInterface.ERROR;
					// write down some info?
				ELSIF (s_fbSeqDockingInterface.q_tmStepTime >= i_stSettings.tClampsTimeout) THEN
 					s_eSeqDockingInterface := E_SeqDockingInterface.ERROR;
					// write down some info?
				END_IF
			
			E_SeqDockingInterface.DOCKING_UNLOCK_DOOR:
			
				IF s_fbSeqDockingInterface.q_bStaEntry THEN 
					s_cmUnlockingPins.m_Unlock();
				END_IF
				
				IF s_cmUnlockingPins.p_bStaIsUnlocked THEN
					s_eSeqDockingInterface := E_SeqDockingInterface.DOCKING_DONE;
				ELSIF s_cmUnlockingPins.p_bStaError THEN 
					s_eSeqDockingInterface := E_SeqDockingInterface.ERROR;
					// write down some info?
				ELSIF (s_fbSeqDockingInterface.q_tmStepTime >= i_stSettings.tReleasePinsTimeout) THEN
 					s_eSeqDockingInterface := E_SeqDockingInterface.ERROR;
					// write down some info?
				END_IF
			
			E_SeqDockingInterface.DOCKING_DONE:
				s_bStaDockingDone := TRUE;
				s_eSeqDockingInterface := E_SeqDockingInterface.IDLE;
			
			E_SeqDockingInterface.UNDOCKING_LOCK_DOOR:
			
				IF s_fbSeqDockingInterface.q_bStaEntry THEN 
					s_cmUnlockingPins.m_Lock();
				END_IF
				
				IF s_cmUnlockingPins.p_bStaIsLocked THEN
					s_eSeqDockingInterface := E_SeqDockingInterface.UNDOCKING_OPEN_CLAMPS;
				ELSIF s_cmUnlockingPins.p_bStaError THEN 
					s_eSeqDockingInterface := E_SeqDockingInterface.ERROR;
					// write down some info?
				ELSIF (s_fbSeqDockingInterface.q_tmStepTime >= i_stSettings.tReleasePinsTimeout) THEN
 					s_eSeqDockingInterface := E_SeqDockingInterface.ERROR;
					// write down some info?
				END_IF
				
			E_SeqDockingInterface.UNDOCKING_OPEN_CLAMPS:
			
				IF s_fbSeqDockingInterface.q_bStaEntry THEN 
					s_cmDockingClamps.m_Open();
				END_IF
				
				IF s_cmDockingClamps.p_bStaIsOpened THEN
					s_eSeqDockingInterface := E_SeqDockingInterface.UNDOCKING_DONE;
				ELSIF s_cmDockingClamps.p_bStaError THEN 
					s_eSeqDockingInterface := E_SeqDockingInterface.ERROR;
					// write down some info?
				ELSIF (s_fbSeqDockingInterface.q_tmStepTime >= i_stSettings.tClampsTimeout) THEN
 					s_eSeqDockingInterface := E_SeqDockingInterface.ERROR;
					// write down some info?
				END_IF
				
			E_SeqDockingInterface.UNDOCKING_DONE:
				s_bStaUndockingDone := TRUE;
				s_eSeqDockingInterface := E_SeqDockingInterface.IDLE;
				
			E_SeqDockingInterface.ONLY_CLOSE_CLAMPS:
			
				IF s_fbSeqDockingInterface.q_bStaEntry THEN
					s_cmDockingClamps.m_Close();
				END_IF
			
				IF s_cmDockingClamps.p_bStaIsClosed THEN
					s_eSeqDockingInterface := E_SeqDockingInterface.IDLE;
				ELSIF (s_fbSeqDockingInterface.q_tmStepTime >= i_stSettings.tClampsTimeout) THEN
 					s_eSeqDockingInterface := E_SeqDockingInterface.ERROR;
					// write down some info?
				END_IF
			
			E_SeqDockingInterface.ONLY_OPEN_CLAMPS:	
				
				IF s_fbSeqDockingInterface.q_bStaEntry THEN
					s_cmDockingClamps.m_Open();
				END_IF
			
				IF s_cmDockingClamps.p_bStaIsOpened THEN
					s_eSeqDockingInterface := E_SeqDockingInterface.IDLE;
				ELSIF (s_fbSeqDockingInterface.q_tmStepTime >= i_stSettings.tClampsTimeout) THEN
 					s_eSeqDockingInterface := E_SeqDockingInterface.ERROR;
					// write down some info?
				END_IF
				
			E_SeqDockingInterface.READY:
				;
			
			E_SeqDockingInterface.ERROR:
				
				IF i_bCmdReset THEN
					//Reset errors (probebly alredy done in the methode devices)
					//--cmValveDockingClampsUpper.i_bCmdReset := TRUE;
				
					s_eSeqDockingInterface := E_SeqDockingInterface.IDLE;
				END_IF
				
		END_CASE		
*)	
		
	E_CtrlMode.MANUAL:
		s_eSeqLiftingTransport := E_SeqTransport.IDLE;
	
		//++_m_ManualControl();
		
//--		// Manual control placed inside the lower layer control modles
	
		{warning '#TODO: Add manual control from hmi'}
		//Is het de bedoeling om op deze plekken de hmi knoppen aan te sturen, OF moet dat gedaan worden in METHOD hmi?		
(*		s_fbHmiBtnManualConveyorApplyBrake.p_bStaVisible := TRUE;
		s_fbHmiBtnManualConveyorApplyBrake.p_bStaEnabled := s_cmPalletConveyor.p_bStaMotorStopped;
	
		s_fbHmiBtnManualConveyorReleaseBrake.p_bStaVisible := TRUE;
		s_fbHmiBtnManualConveyorReleaseBrake.p_bStaEnabled := s_cmPalletConveyor.p_bStaMotorStopped;
		
		s_fbHmiBtnManualConveyorStop.p_bStaVisible := TRUE;
		s_fbHmiBtnManualConveyorStop.p_bStaEnabled := TRUE;
	
		s_fbHmiBtnManualConveyorForward.p_bStaVisible := TRUE;
		s_fbHmiBtnManualConveyorForward.p_bStaEnabled := s_cmPalletConveyor.p_bStaMotorStopped;
	
		s_fbHmiBtnManualConveyorBackward.p_bStaVisible := TRUE;
		s_fbHmiBtnManualConveyorBackward.p_bStaEnabled := s_cmPalletConveyor.p_bStaMotorStopped;
		
		IF s_fbHmiBtnManualConveyorApplyBrake.p_osrBtnPress THEN
			s_cmPalletConveyor.m_ReleaseBrake(i_bValue := FALSE);
		END_IF
		
		IF s_fbHmiBtnManualConveyorReleaseBrake.p_osrBtnPress THEN
			s_cmPalletConveyor.m_ReleaseBrake(i_bValue := TRUE);
		END_IF
	
		IF s_fbHmiBtnReset.p_osrBtnPress THEN
			s_cmPalletConveyor.m_Reset();
		END_IF
			
		IF s_fbHmiBtnManualConveyorStop.p_osrBtnPress THEN
			s_cmPalletConveyor.m_Stop();	
		ELSIF s_fbHmiBtnManualConveyorForward.p_osrBtnPress THEN
			s_cmPalletConveyor.m_StartForward(i_rTargetSpeed := i_stSettings.rSpeedManual);
		ELSIF s_fbHmiBtnManualConveyorBackward.p_osrBtnPress THEN
			s_cmPalletConveyor.m_StartBackward(i_rTargetSpeed := i_stSettings.rSpeedManual);
		END_IF
*)		
END_CASE

m_Main := TRUE;
END_METHOD

{attribute 'TcRpcEnable'}
METHOD PUBLIC m_ReqCenteringTB : BOOL

IF NOT i_bReqEnable THEN 
	RETURN;
END_IF

IF NOT i_bReqEnable THEN 
	RETURN;
END_IF

s_bReqCenteringTB := TRUE;

m_ReqCenteringTB := TRUE;
END_METHOD

{attribute 'TcRpcEnable'}
METHOD PUBLIC m_ReqTB_ToCenter : BOOL

IF NOT i_bReqEnable THEN 
	RETURN;
END_IF

s_bReqTB_ToCenter := TRUE;

m_ReqTB_ToCenter := TRUE;
END_METHOD

{attribute 'TcRpcEnable'}
METHOD PUBLIC m_ReqTB_ToDocking : BOOL

IF NOT i_bReqEnable THEN 
	RETURN;
END_IF

s_bReqTB_ToDocking := TRUE;

m_ReqTB_ToDocking := TRUE;
END_METHOD

{attribute 'TcRpcEnable'}
METHOD PUBLIC m_ReqTB_ToInfeed : BOOL

IF NOT i_bReqEnable THEN 
	RETURN;
END_IF

s_bReqTB_ToInfeed := TRUE;

m_ReqTB_ToInfeed := TRUE;
END_METHOD

PROPERTY PUBLIC p_bStaTB_AtCentering : BOOL
GET

p_bStaTB_AtCentering := s_bStaTB_AtCentering;
END_GET
END_PROPERTY

PROPERTY PUBLIC p_bStaTB_AtDocking : BOOL
GET

p_bStaTB_AtDocking := s_bStaTB_AtDocking;
END_GET
END_PROPERTY

PROPERTY PUBLIC p_bStaTB_AtInfeed : BOOL
GET

p_bStaTB_AtInfeed := s_bStaTB_AtInfeed;
END_GET
END_PROPERTY

PROPERTY PUBLIC p_bStaTB_CenteringDone : BOOL
GET

p_bStaTB_CenteringDone := s_bStaTB_CenteringDone;
END_GET
END_PROPERTY

END_FUNCTION_BLOCK

(* stored: Version 1.1.0.1, ProductVersion 3.1.4024.12
   POU EM_LiftingTransport: Id {82ac1e56-2937-4df1-886d-5bc6dc15361f}, SpecialFunc None
   Method _m_Alarms: Id {77ac2c1c-b354-4acb-9f0d-e0fd9e0a3a94}
   Method _m_AutomaticControl: Id {51dbf1d4-9c3c-42ad-87fe-cdadd1984100}
   Method _m_Devices: Id {b95b1090-f72e-49a8-b75a-87fbc22bb2f7}
   Method _m_Hmi: Id {86cd5a15-a053-432c-9e95-504bd0cfab5b}
   Method _m_Init: Id {fdcbf52e-0860-4b94-915e-8e7c2bbd0a27}
   Method _m_Inputs: Id {2c09f905-698a-4dfd-8c60-1a7d7f6d646b}
   Method _m_ManualControl: Id {61a84643-dbec-4bc1-99bd-3a2ec3342898}
   Method _m_MoveAbsolute: Id {7f8f7561-70c1-4897-9a57-d3b7b8c51729}
   Method _m_Outputs: Id {0027b51b-0e3b-4c47-b79c-c262d8cada1b}
   Method _m_Params: Id {5f8e46d4-1bd2-48a0-a796-5af6a0b2577f}
   Method _m_SeqLiftingTransport: Id {adfb5128-2b00-4a29-b7de-b50ba035879a}
   Method m_CmdCenteringTB: Id {5f07294c-c083-4786-a1a2-586c95e439f7}
   Method m_CmdTB_ToCenter: Id {3a534c15-c636-468b-8b82-6fd59e761d1a}
   Method m_CmdTB_ToDocking: Id {fddfe49e-6281-47a3-8534-8abf984608e2}
   Method m_CmdTB_ToInfeed: Id {05a177ec-65c8-4b07-91b0-bc7997926449}
   Method m_Main: Id {7d708d4c-1fee-4511-a8d0-db3dbe3fd7e6}
   Method m_ReqCenteringTB: Id {415ce6ea-afb8-4118-a1fc-ea58b530d7b6}
   Method m_ReqTB_ToCenter: Id {9d30bbef-bcd6-4fc2-8d93-9b2201ca737f}
   Method m_ReqTB_ToDocking: Id {bc26af41-4ec1-4049-ae2f-a8f4c7a26c9b}
   Method m_ReqTB_ToInfeed: Id {fa516528-012b-4031-8e18-317ece30b039}
   Property p_bStaTB_AtCentering: Id {050383f4-1821-4a98-ab50-f2e654340431}
   Get Get: Id {03f3f379-9c7e-473c-8407-742758c9f4b6}
   Property p_bStaTB_AtDocking: Id {630d4760-3c9e-490a-b1db-ceb84ce3b93d}
   Get Get: Id {ac0f1cfe-6ddb-4648-8ead-590b388c0171}
   Property p_bStaTB_AtInfeed: Id {ccba55b7-671b-48a2-af2d-7bdd569222c9}
   Get Get: Id {c55ed7dc-3eae-49e0-bba0-c67b4ed5fb10}
   Property p_bStaTB_CenteringDone: Id {92f12f64-9c7b-449f-90f0-528b8c0b82e0}
   Get Get: Id {f8e455bd-3d78-46ed-aec1-a530ae8bd329} *)
